PROGRAM CraneSimulation
VAR
	fTime : LREAL; 	
	bRunning : BOOL;
	fPositionAutoMode : LREAL; 
	fInitialPosition : LREAL; 
	fInitialVelocity : LREAL; 
END_VAR

IF Inputs.bStartSimulation AND Inputs.bAutoMode  THEN
	fTime := fTime + Parameters.fCyclicTime;
ELSE
	fTime := 0; 	
END_IF

IF fTime > 0 AND Inputs.bAutoMode THEN 
	bRunning := TRUE;
ELSE
	bRunning := FALSE;
END_IF

fPositionAutoMode := Inputs.fCylinderVelocityReference * (fTime * fTime)/2 + fInitialVelocity * fTime + fInitialPosition;

//IF fPositionAutoMode >= 1 THEN
//	Outputs.fCylinderPosition := 1;	
//ELSIF fPosition <= 0 THEN
//	Outputs.fCylinderPosition := 0; 
//ELSE	
//	Outputs.fCylinderPosition := fPositionAutoMode;
//END_IF

IF Inputs.bAutoMode THEN
	Outputs.fCylinderPosition := fPositionAutoMode;
ELSE
	Outputs.fCylinderPosition := Inputs.fManualCylinderPositionReference;	
END_IF

Outputs.bSimulationRunning := bRunning;  
Outputs.fSimulationTime := fTime; 
Outputs.fCylinderVelocity := Inputs.fCylinderVelocityReference;
Outputs.pt1_y := LREAL_TO_INT(Outputs.fCylinderPosition * Parameters.fPistonScale);

END_PROGRAM

(* stored: Version 1.1.0.1, ProductVersion 3.1.4024.10
   POU CraneSimulation: Id {c255987f-7a58-4573-9ac9-545c12e8d4a5}, SpecialFunc None *)
